PROGRAM PickandPlace
VAR
END_VAR

END_PROGRAM

(* stored: Version 1.1.0.1, ProductVersion 3.1.4024.15
   POU PickandPlace: Id {bf1217fb-f291-4d9f-ad63-4b91b16f2452}, SpecialFunc None *)
